Fanuc KAREL source: IO0118.KL

PROGRAM IO0118
%STACKSIZE=65535
%PRIORITY=65535
%NOLOCKGROUP
ROUTINE RTEST FROM IO0118
ROUTINE RTEST
VAR
L1 : ARRAY[3] OF INTEGER
L2 : XYZWPR
L3 : JOINTPOS9
L4 : POSITION
U2C_37 : INTEGER
U2C_38 : REAL
U2C_39 : REAL
U2C_40 : INTEGER
U2C_41 : REAL
BEGIN
U2C_37=1
L1[1]=2
U2C_40=1
U2C_41=1.0
-- UNSAFE_SOURCE_IR line 19: FRAME[RTEST+0x28] = native_io_value(9, (FRAME[RTEST+0x25] + 1))
END RTEST
BEGIN
RTEST
END IO0118
